// TIA Portal V18 export
DATA_BLOCK "MC_MoveJog_DB"   // DB21
// stored: AutoNumber true, DBAccessibleFromOPCUA true, InstanceOfName MC_MoveJog, OfSystemLibElement MC_MoveJog, OfSystemLibVersion 7.0
"MC_MoveJog"
   // VAR_INPUT
   //    Axis : TO_SpeedAxis;
   //    JogForward : Bool;
   //    JogBackward : Bool;
   //    Velocity : Real;
   //    PositionControlled : Bool;
   // END_VAR
   // VAR_OUTPUT
   //    InVelocity : Bool;
   //    Busy : Bool;
   //    CommandAborted : Bool;
   //    Error : Bool;
   //    ErrorID : Word;
   //    ErrorInfo : Word;
   // END_VAR
   // VAR
   //    FB_ID : DInt;
   // END_VAR
BEGIN
END_DATA_BLOCK
